Staubli VAL3: VelocityAddon.pjx

--- VelocityAddon.pjx ---
Parameters version=s7.8 stackSize=5000 millimeterUnit=true
Program file=setVel.pgx
Program file=start.pgx
Program file=stop.pgx
Data file=VelocityAddon.dtx

--- VelocityAddon.dtx ---
mdesc mNomSpeed
bool bSync
mdesc mNominal = {tmax=100, rmax=100, leave=1, reach=1, blend=cartesian}
tool tTool = {fatherId=flange[0], ioLink=valve1}
num nVelCmd[6]
num nMoveType

--- start.pgx ---
program start()
begin
  //nMoveType:
  //0:Frame
  //1:tool
  //2:joint
  taskCreateSync "vel",0.004,bSync,setVel(nMoveType,world,tTool,mNominal,nVelCmd)
end

--- setVel.pgx ---
program setVel(num x_nVelType, frame x_fVelFrm, tool x_tTool, mdesc x_mMdesc, num& x_nCmd[])
  local num l_ni
begin
  //choose the type
  switch x_nVelType
    case 1
      $velTool(x_tTool,x_mMdesc)
    break
    case 2
      $velJoint(x_tTool,x_mMdesc)
    break
    default
      $velFrame(x_fVelFrm,x_tTool,x_mMdesc)
    break
  endSwitch
  //
  while true
    $setVelCmd(x_nCmd)
    delay(0)
  endWhile
end
